FUNCTION_BLOCK FB_TextReport EXTENDS FB_TestReportBase

(******************************************************************************
Baustein: FB_TestReportBase.BuildFile
Spezifikation: doc/Spezifikation.pdf, Kap. x.y.z
-------------------------------------------------------------------------------
erstellt:
von:
Geändert:
von:
-------------------------------------------------------------------------------
Beschreibung
Diese Methode muss vom ableitenden Baustein überschrieben werden und
wird von der Basisklasse aus aufgerufen wenn der Report erstellt werden
soll.

-------------------------------------------------------------------------------
Input
-

Output
-
******************************************************************************)
METHOD PROTECTED BuildFile : ERetCode_t
VAR_INPUT
	i_u32Line : UDINT;
END_VAR

	BuildFile := ERetCode_t.eRetBusy;

	CASE i_u32Line OF

	0: addString('Test Report :');
	   addDate(getTime());
	   addString(' - ');
	   addTime(getTime());
	1: addString('++++++++++++++++++++++++++++++++++++++++++++++++++');
	2: //
	3: //

	4: addString('Asserts gesamt: ');
	   addValue(sStatistic.u32Asserts);

	5: addString('Asserts passed: ');
	   addValue(sStatistic.u32Passed);

	6: addString('Asserts failed: ');
	   addValue(sStatistic.u32Failed);

	7: //

	9:  addString('Ergebnis : ');
		IF sStatistic.u32Failed > 0 THEN
			addString('FAILED');
		ELSE
			addString('PASSED');
		END_IF;

	10: addString('++++++++++++++++++++++++++++++++++++++++++++++++++');
	
	99: BuildFile := ERetCode_t.eRetDone;

	END_CASE;
END_METHOD

(******************************************************************************
Baustein: FB_TestReportBase.getFileName
Spezifikation: doc/Spezifikation.pdf, Kap. x.y.z
-------------------------------------------------------------------------------
erstellt:
von:
Geändert:
von:
-------------------------------------------------------------------------------
Beschreibung
Diese Methode muss vom ableitenden Baustein überschrieben werden und
wird von der Basisklasse aus aufgerufen wenn der Report erstellt werden
soll.

-------------------------------------------------------------------------------
Input
-

Output
-
******************************************************************************)
METHOD PROTECTED getFileName : ERetCode_t
VAR_INPUT
	i_pFileName : NameHandle_t;
	i_pPath		: PathHandle_t;
END_VAR
VAR
	sTime : TIMESTRUCT;
END_VAR

	i_pFileName^ := 'Exp_';
	i_pPath^ 	 := 'C:\Users\Administrator\Desktop\TestResult\';

	sTime := getTime();

	i_pFileName^ := Concat(i_pFileName^, WORD_TO_STRING(sTime.wYear));
	i_pFileName^ := Concat(i_pFileName^, DWORD_TO_DECSTR(sTime.wMonth, 2));
	i_pFileName^ := Concat(i_pFileName^, DWORD_TO_DECSTR(sTime.wDay  , 2));
	i_pFileName^ := Concat(i_pFileName^, '_');
	i_pFileName^ := Concat(i_pFileName^, DWORD_TO_DECSTR(sTime.wHour  , 2));
	i_pFileName^ := Concat(i_pFileName^, DWORD_TO_DECSTR(sTime.wMinute, 2));
	i_pFileName^ := Concat(i_pFileName^, '.txt');
END_METHOD

END_FUNCTION_BLOCK

(* stored: Version 1.1.0.1, ProductVersion 3.1.4024.13
   POU FB_TextReport: Id {3b012d41-7e00-4335-8587-d56a2a32ec42}, SpecialFunc None
   Method BuildFile: Id {fc563d74-bc6f-4dab-994a-1845441da6c6}
   Method getFileName: Id {781f0045-a5e7-4897-bc3c-2f4f70da5c1c} *)
